// TIA Portal project "learning100" (V20)

(* hardware
DEVICE "S7-1200 station_1"  S7-1200 Station
   slot 0: "Rack_0"  S7-1200 Rack  Rack  V1.0
   slot 1: "PLC_1"  CPU 1212FC DC/DC/RLY  6ES7 212-1HF40-0XB0  V4.7
DEVICE "HMI_1"  KTP700 Basic DP
   slot 0: "HMI_1"  KTP700 Basic DP  6AV2 123-2GA03-0AX0  17.0.0.0
   slot 1: "HMI_RT_1"  KTP700 Basic DP  6AV2 123-2GA03-0AX0  17.0.0.0
   slot 7: "HMI_1.MPI/DP_CP_1"  MPI/DP Interface  17.0.0.0
*)

// ===== PLC "PLC_1"  CPU 1212FC DC/DC/RLY =====

VAR_GLOBAL   // PLC tag table "Default tag table"
   "pushbutton1" AT %M0.0 : Bool;
   "pushbutton2" AT %M0.1 : Bool;
   "LED1" AT %M0.2 : Bool;
   "LED2" AT %M0.3 : Bool;
END_VAR

DATA_BLOCK "Main_Safety_RTG1_DB"   // DB1, F_DB
{ S7_Optimized_Access := 'TRUE' }
NAME : FUSI
VERSION : 0.1
// stored: InstanceOfName Main_Safety_RTG1
"Main_Safety_RTG1"
BEGIN
END_DATA_BLOCK

FUNCTION_BLOCK "Main_Safety_RTG1"   // FB1, F_FBD
{ S7_Optimized_Access := 'TRUE' }
BEGIN
END_FUNCTION_BLOCK

ORGANIZATION_BLOCK "Main"   // OB1, LAD, ProgramCycle
TITLE = "Main Program Sweep (Cycle)"
{ S7_Optimized_Access := 'TRUE' }
VERSION : 0.1
   VAR_INPUT
      Initial_Call : Bool;   // Initial call of this OB
      Remanence : Bool;   // =True, if remanent data are available
   END_VAR
BEGIN

REGION Network 1
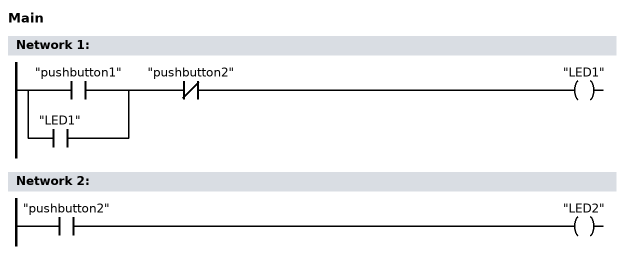
   RUNG wire#powerrail
      Contact( "pushbutton1" )
      wire#w1
      I_Contact( "pushbutton2" )
      Coil( "LED1" )
   END_RUNG
   RUNG wire#powerrail
      Contact( "LED1" )
   END_RUNG wire#w1
   // the same network as SCL:
   "LED1" := ("pushbutton1" OR "LED1") AND NOT "pushbutton2";
END_REGION

REGION Network 2
   RUNG wire#powerrail
      Contact( "pushbutton2" )
      Coil( "LED2" )
   END_RUNG
   // the same network as SCL:
   "LED2" := "pushbutton2";
END_REGION
END_ORGANIZATION_BLOCK

(* ===== HMI "HMI_RT_1" =====
system functions are stored by id; their names below are inferred from use
connection "HMI_Connection_1": IF1 B, SMART_S7_1200_OMS

HMI tags "Default tag table"
   "PUSHBUTTON1" : Bool = PLC pushbutton1 AT %M0.0, 1 s
   "PUSHBUTTON2" : Bool = PLC pushbutton2 AT %M0.1, 1 s
   "LED1" : Bool = PLC LED1 AT %M0.2, 1 s
   "LED2" : Bool = PLC LED2 AT %M0.3, 1 s

Template "Template_1" 800x480
   Button "Exit" at 714,429 size 71x50; TextOff 'Exit'; PictureOff "ExitRuntime_KTP700_Basic_DP_TR"; PictureOn "ExitRuntime_KTP700_Basic_DP_TR"
      on Release: StopRuntime(0)
   Button "Template_Button" at 614,429 size 71x50; TextOff 'Text'
   Button "Template_Button_1" at 514,429 size 71x50; TextOff 'Text'
   Button "Template_Button_2" at 414,429 size 71x50; TextOff 'Text'
   Button "Template_Button_3" at 314,429 size 71x50; TextOff 'Text'
   Button "Template_Button_4" at 214,429 size 71x50; TextOff 'Text'
   Button "Template_Button_5" at 114,429 size 71x50; TextOff 'Text'
   Button "Start screen" at 14,429 size 71x50; TextOff 'Start screen'; PictureOff "NavigateHome_KTP700_Basic_DP_TR"; PictureOn "NavigateHome_KTP700_Basic_DP_TR"
      on Release: ActivateScreen("Root screen", 0)
   SymbolicIOField "Symbolic_IO_Field_Screen" at 93,9 size 600x33; TextOff '0'; TextOn '1'; TextList "TextList_ScreenNames"
      ProcessValue <- "Tag_ScreenNumber"
      on Change: ActivateScreenByNumber("Tag_ScreenNumber", 0)
   DateTimeField "HmiScreenItemData" at 695,25 size 105x25
   DateTimeField "HmiScreenItemData_1" at 695,0 size 105x25
   GraphicView "Logo" at 0,0 size 91x51; Picture "Logo of HMI_1"

screen "Root screen" 800x480, template "Template_1"
   on GenerateScreen: SetTag("Tag_ScreenNumber", 1)
   Button "Button_1" at 56,260 size 96x32; TextOff 'PB1'
      on Press: SetBit("PUSHBUTTON1")
      on Release: ResetBit("PUSHBUTTON1")
   Button "Button_2" at 57,306 size 96x32; TextOff 'PB2'
      on Press: SetBit("PUSHBUTTON2")
      on Release: ResetBit("PUSHBUTTON2")
   Circle "Circle_1" at 231,251 size 48x48
      Appearance <- "LED1"
   Circle "Circle_2" at 230,306 size 48x48
      Appearance <- "LED2"
*)